FUNCTION_BLOCK SET_STRUCT_VALUE (* Service Interface Function Block Type *)
  (* Standard: 61499-2; Description: Copyright (c) 2023 Primetals Technologies Austria GmbH This program and the accompanying materials are made available under the terms of the Eclipse Public License 2.0 which is available at https://www.eclipse.org/legal/epl-2.0/ SPDX-License-Identifier: EPL-2.0 *)
  (* Version 1.0, 2023-03-06, Alois Zoitl *)
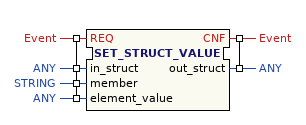
  EVENT_INPUT
    REQ WITH member, in_struct, element_value; (* Set Value out of structure *)
  END_EVENT
  EVENT_OUTPUT
    CNF WITH out_struct; (* REQ event finished *)
  END_EVENT
  VAR_INPUT
    in_struct : ANY; (* Structure to look into *)
    member : STRING; (* Member of the strucuture to retrieve. Inner members are access using the dot (.) operator *)
    element_value : ANY; (* new value for the element *)
  END_VAR
  VAR_OUTPUT
    out_struct : ANY; (* TRUE if no errors ocurred, FALSE otherwise *)
  END_VAR
END_FUNCTION_BLOCK
